TYPE ST_BaseLoggerElement_HMI :
STRUCT
	refstMemoryEvents				: REFERENCE TO ST_BaseEvents_Memory;
	
END_STRUCT
END_TYPE

(* stored: Version 1.1.0.1
   DUT ST_BaseLoggerElement_HMI: Id {0ce980ad-4c50-07a7-0c2d-226937f06ada} *)
